// TIA Portal V18 export
FUNCTION "Flowrate adjustment configuration B" : Void   // FC10, LAD
{ S7_Optimized_Access := 'TRUE' }
VERSION : 0.1
// stored: AutoNumber false, IsIECCheckEnabled false, SetENOAutomatically false, UDAEnableTagReadback false
BEGIN

REGION Network 1 (SCL)
   IF "Pump & Flowrate"."Calculated Flowrate B without adjustment" <= "Pump & Flowrate".capacity."pump B" * 0.05 THEN
       "Pump & Flowrate"."fowrate B Adjustment Configuration" := "Flowrate adjustment B".percentage."5%";
   ELSIF "Pump & Flowrate"."Calculated Flowrate B without adjustment" <= "Pump & Flowrate".capacity."pump B" * 0.10 THEN
       "Pump & Flowrate"."fowrate B Adjustment Configuration" := "Flowrate adjustment B".percentage."10%";
   ELSIF "Pump & Flowrate"."Calculated Flowrate B without adjustment" <= "Pump & Flowrate".capacity."pump B" * 0.15 THEN
       "Pump & Flowrate"."fowrate B Adjustment Configuration" := "Flowrate adjustment B".percentage."15%";
   ELSIF "Pump & Flowrate"."Calculated Flowrate B without adjustment" <= "Pump & Flowrate".capacity."pump B" * 0.20 THEN
       "Pump & Flowrate"."fowrate B Adjustment Configuration" := "Flowrate adjustment B".percentage."20%";
   ELSIF "Pump & Flowrate"."Calculated Flowrate B without adjustment" <= "Pump & Flowrate".capacity."pump B" * 0.25 THEN
       "Pump & Flowrate"."fowrate B Adjustment Configuration" := "Flowrate adjustment B".percentage."25%";
   ELSIF "Pump & Flowrate"."Calculated Flowrate B without adjustment" <= "Pump & Flowrate".capacity."pump B" * 0.30 THEN
       "Pump & Flowrate"."fowrate B Adjustment Configuration" := "Flowrate adjustment B".percentage."30%";
   ELSIF "Pump & Flowrate"."Calculated Flowrate B without adjustment" <= "Pump & Flowrate".capacity."pump B" * 0.40 THEN
       "Pump & Flowrate"."fowrate B Adjustment Configuration" := "Flowrate adjustment B".percentage."40%";
   ELSIF "Pump & Flowrate"."Calculated Flowrate B without adjustment" <= "Pump & Flowrate".capacity."pump B" * 0.50 THEN
       "Pump & Flowrate"."fowrate B Adjustment Configuration" := "Flowrate adjustment B".percentage."50%";
   ELSIF "Pump & Flowrate"."Calculated Flowrate B without adjustment" <= "Pump & Flowrate".capacity."pump B" * 0.60 THEN
       "Pump & Flowrate"."fowrate B Adjustment Configuration" := "Flowrate adjustment B".percentage."60%";
   ELSIF "Pump & Flowrate"."Calculated Flowrate B without adjustment" <= "Pump & Flowrate".capacity."pump B" * 0.70 THEN
       "Pump & Flowrate"."fowrate B Adjustment Configuration" := "Flowrate adjustment B".percentage."70%";
   ELSIF "Pump & Flowrate"."Calculated Flowrate B without adjustment" <= "Pump & Flowrate".capacity."pump B" * 0.80 THEN
       "Pump & Flowrate"."fowrate B Adjustment Configuration" := "Flowrate adjustment B".percentage."80%";
   ELSIF "Pump & Flowrate"."Calculated Flowrate B without adjustment" <= "Pump & Flowrate".capacity."pump B" * 0.90 THEN
       "Pump & Flowrate"."fowrate B Adjustment Configuration" := "Flowrate adjustment B".percentage."90%";
   ELSE
       "Pump & Flowrate"."fowrate B Adjustment Configuration" := "Flowrate adjustment B".percentage."100%";
   END_IF;
END_REGION

REGION Network 2: reset alladjustment
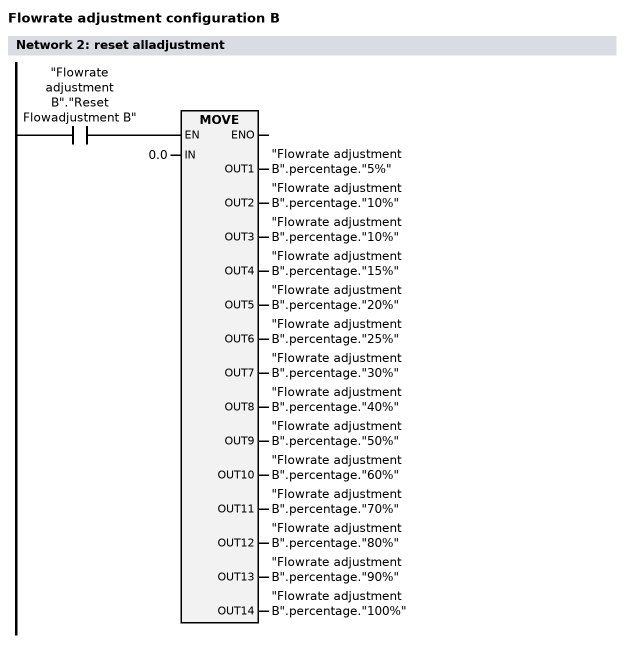
   RUNG wire#powerrail
      Contact( "Flowrate adjustment B"."Reset Flowadjustment B" )
      Move(in := 0.0, out1 => "Flowrate adjustment B".percentage."5%", out2 => "Flowrate adjustment B".percentage."10%", out3 => "Flowrate adjustment B".percentage."10%", out4 => "Flowrate adjustment B".percentage."15%", out5 => "Flowrate adjustment B".percentage."20%", out6 => "Flowrate adjustment B".percentage."25%", out7 => "Flowrate adjustment B".percentage."30%", out8 => "Flowrate adjustment B".percentage."40%", out9 => "Flowrate adjustment B".percentage."50%", out10 => "Flowrate adjustment B".percentage."60%", out11 => "Flowrate adjustment B".percentage."70%", out12 => "Flowrate adjustment B".percentage."80%", out13 => "Flowrate adjustment B".percentage."90%", out14 => "Flowrate adjustment B".percentage."100%")
   END_RUNG
   // the same network as SCL:
   IF "Flowrate adjustment B"."Reset Flowadjustment B" THEN
       "Flowrate adjustment B".percentage."5%" := 0.0;
       "Flowrate adjustment B".percentage."10%" := 0.0;
       "Flowrate adjustment B".percentage."10%" := 0.0;
       "Flowrate adjustment B".percentage."15%" := 0.0;
       "Flowrate adjustment B".percentage."20%" := 0.0;
       "Flowrate adjustment B".percentage."25%" := 0.0;
       "Flowrate adjustment B".percentage."30%" := 0.0;
       "Flowrate adjustment B".percentage."40%" := 0.0;
       "Flowrate adjustment B".percentage."50%" := 0.0;
       "Flowrate adjustment B".percentage."60%" := 0.0;
       "Flowrate adjustment B".percentage."70%" := 0.0;
       "Flowrate adjustment B".percentage."80%" := 0.0;
       "Flowrate adjustment B".percentage."90%" := 0.0;
       "Flowrate adjustment B".percentage."100%" := 0.0;
   END_IF;
END_REGION
END_FUNCTION
